Universal Robots URScript: set_b_draw_borders.bak.script

def set_b_draw_bordersbak():
  set_tcp(p[0.0,0.0,0.0,0.0,0.0,0.0])
  set_safety_mode_transition_hardness(1)
  set_tool_communication(True, 1000000, 2, 1, 1.5, 3.5)
  set_tool_output_mode(0)
  set_tool_digital_output_mode(0, 1)
  set_tool_digital_output_mode(1, 1)
  set_tool_voltage(0)
  step_count_92a71080_320b_48c3_b710_fb27a0ae3266 = 0.0
  thread Step_Counter_Thread_29a6b4c0_57cd_4359_a365_f92f2370702e():
    while (True):
      step_count_92a71080_320b_48c3_b710_fb27a0ae3266 = step_count_92a71080_320b_48c3_b710_fb27a0ae3266 + 1.0
      sync()
    end
  end
  run Step_Counter_Thread_29a6b4c0_57cd_4359_a365_f92f2370702e()
  set_gravity([0.0, 0.0, 9.82])
  set_standard_analog_input_domain(0, 1)
  set_standard_analog_input_domain(1, 1)
  set_tool_analog_input_domain(0, 1)
  set_tool_analog_input_domain(1, 1)
  set_analog_outputdomain(0, 0)
  set_analog_outputdomain(1, 0)
  set_input_actions_to_default()
  set_target_payload(1.070000, [0.002000, 0.003000, 0.057000], [0.001723, 0.001723, 0.001723, 0.000000, 0.000000, 0.000000])
  global Plane_1=p[-0.700006141123905,1.3454883874109249E-6,0.3910559577028425,-1.2089868272251132,-1.2089999932245832,1.20858562628424]
  global Plane_2=p[0.0,0.0,0.0,0.0,0.0,0.0]
  global Point_1=p[0.6913645118948067,-0.12399382748223003,0.49223711947071,-1.2983729986843258,1.1259514972191385,-1.2203503861141718]
  $ 1 "Robot Program"
  $ 2 "Script: draw_borders.script"
  def Machining3():
    # Default parameters:
    global speed_ms = 0.3
    global speed_rads = 0.75
    global accel_mss = 3
    global accel_radss = 1.2
    global blend_radius_m = 0.001

    # Add subprograms here
    # Start of main program
    # Program generated by RoboDK v5.6.5 for UR10e on 17/10/2023 11:41:04
    # Using nominal kinematics.
    blend_radius_m = 0.001
    speed_ms = 1.000
    # set_reference(p[0.335000, -0.154000, -0.015800, 0.000000, 0.000000, 0.000000])
    set_tcp(p[0.000000, 0.000000, 0.252000, 0.000000, 0.000000, 0.000000])
    # Show Tool
    movej([0.061043, -1.073805, -2.582860, -1.055724, 1.570796, 1.631840],accel_radss,speed_rads,0,blend_radius_m)
    movel([0.061043, -1.164815, -2.648932, -0.898642, 1.570796, 1.631840],accel_mss,speed_ms,0,blend_radius_m)
    speed_ms = 1.000
    speed_ms = 0.005
    movel([0.061043, -1.124589, -2.623317, -0.964483, 1.570796, 1.631840],accel_mss,speed_ms,0,blend_radius_m)
    speed_ms = 1.000
    movel([0.061043, -1.164815, -2.648932, -0.898642, 1.570796, 1.631840],accel_mss,speed_ms,0,blend_radius_m)
    speed_ms = 0.040
    speed_ms = 1.000
    movel([0.157276, -1.127729, -2.665258, -0.919402, 1.570796, 1.728073],accel_mss,speed_ms,0,blend_radius_m)
    speed_ms = 0.005
    movel([0.157276, -1.174031, -2.690432, -0.847927, 1.570796, 1.728073],accel_mss,speed_ms,0,blend_radius_m)
    speed_ms = 0.035
    movel([0.061043, -1.210716, -2.673294, -0.828379, 1.570796, 1.631840],accel_mss,speed_ms,0,blend_radius_m)
    movel([0.051500, -1.358795, -2.587796, -0.765798, 1.570796, 1.622297],accel_mss,speed_ms,0,blend_radius_m)
    movel([0.044558, -1.480296, -2.495031, -0.737062, 1.570796, 1.615354],accel_mss,speed_ms,0,blend_radius_m)
    movel([0.113774, -1.462570, -2.509956, -0.739863, 1.570796, 1.684571],accel_mss,speed_ms,0,blend_radius_m)
    movel([0.183803, -1.448210, -2.521691, -0.742489, 1.570796, 1.754599],accel_mss,speed_ms,0,blend_radius_m)
    movel([0.213690, -1.314067, -2.616588, -0.781734, 1.570796, 1.784487],accel_mss,speed_ms,0,blend_radius_m)
    movel([0.255784, -1.142912, -2.703858, -0.865619, 1.570796, 1.826580],accel_mss,speed_ms,0,blend_radius_m)
    movel([0.157276, -1.174031, -2.690432, -0.847927, 1.570796, 1.728073],accel_mss,speed_ms,0,blend_radius_m)
    movel([0.154107, -1.175144, -2.689933, -0.847312, 1.570796, 1.724904],accel_mss,speed_ms,0,blend_radius_m)
    speed_ms = 0.005
    movel([0.154107, -1.128851, -2.664784, -0.918754, 1.570796, 1.724904],accel_mss,speed_ms,0,blend_radius_m)
    speed_ms = 1.000
    movel([0.154107, -1.038314, -2.596953, -1.077123, 1.570796, 1.724904],accel_mss,speed_ms,0,blend_radius_m)
    # End of main program
  end

  Machining3()
end
